FUNCTION F_Sample : INT
VAR_INPUT
	nVar1 : INT;
	nVar2 : INT;
	nVar3 : INT;
END_VAR
VAR
	FunTemp : INT;
END_VAR

F_Sample := nVar1 + nVar2 +nVar3;

END_FUNCTION

(* stored: Version 1.1.0.1, ProductVersion 3.1.4024.10
   POU F_Sample: Id {b265c7ce-0f94-49c5-94a9-8dcc1578d2ce}, SpecialFunc None *)
